SUBAPPLICATION Uebung_160_AX (* Motor Links/Rechtslauf *)
  (* Standard: 61499-2; Description: Copyright (c) 2023 Meisterschulen am Ostbahnhof This program and the accompanying materials are made available under the terms of the Eclipse Public License 2.0 which is available at https://www.eclipse.org/legal/epl-2.0/ SPDX-License-Identifier: EPL-2.0 *)
  (* Version 1.0, 2023-10-23, Franz Höpfinger, Meisterschulen am Ostbahnhof, initial API and implementation and/or initial documentation *)
  PACKAGE Uebungen;
  IMPORT logiBUS::io::DI::logiBUS_DI::Input_I1;
  IMPORT logiBUS::io::DI::logiBUS_DI::Input_I2;
  IMPORT logiBUS::io::DQ::logiBUS_DO::Output_Q5;
  IMPORT logiBUS::io::DQ::logiBUS_DO::Output_Q56;
  IMPORT logiBUS::io::DQ::logiBUS_DO::Output_Q6;
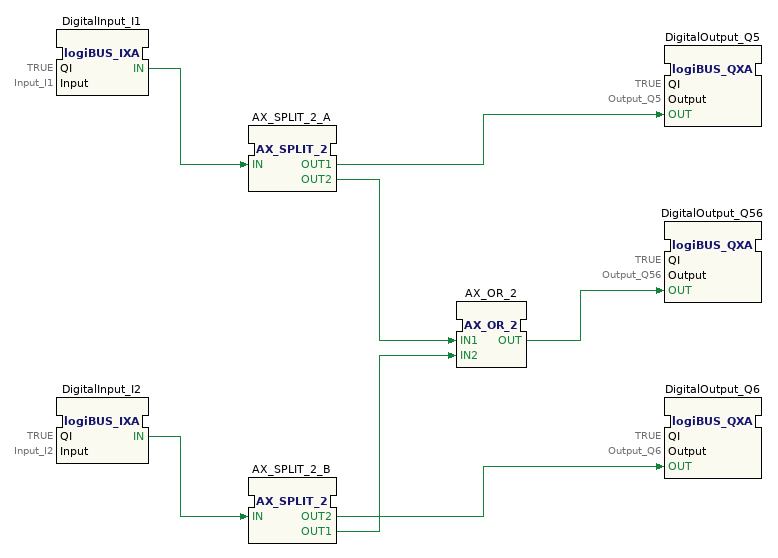
  FBS
    DigitalInput_I1 : logiBUS::io::DI::logiBUS_IXA(QI := TRUE, Input := Input_I1);
    DigitalOutput_Q5 : logiBUS::io::DQ::logiBUS_QXA(QI := TRUE, Output := Output_Q5);
    DigitalOutput_Q6 : logiBUS::io::DQ::logiBUS_QXA(QI := TRUE, Output := Output_Q6);
    DigitalInput_I2 : logiBUS::io::DI::logiBUS_IXA(QI := TRUE, Input := Input_I2);
    AX_OR_2 : adapter::booleanOperators::AX_OR_2;
    DigitalOutput_Q56 : logiBUS::io::DQ::logiBUS_QXA(QI := TRUE, Output := Output_Q56);
    AX_SPLIT_2_A : adapter::events::unidirectional::AX_SPLIT_2;
    AX_SPLIT_2_B : adapter::events::unidirectional::AX_SPLIT_2;
  END_FBS
  ADAPTER_CONNECTIONS
    DigitalInput_I1.IN TO AX_SPLIT_2_A.IN;
    AX_SPLIT_2_A.OUT1 TO DigitalOutput_Q5.OUT;
    DigitalInput_I2.IN TO AX_SPLIT_2_B.IN;
    AX_SPLIT_2_B.OUT2 TO DigitalOutput_Q6.OUT;
    AX_OR_2.OUT TO DigitalOutput_Q56.OUT;
    AX_SPLIT_2_A.OUT2 TO AX_OR_2.IN1;
    AX_SPLIT_2_B.OUT1 TO AX_OR_2.IN2;
  END_CONNECTIONS
END_SUBAPPLICATION
